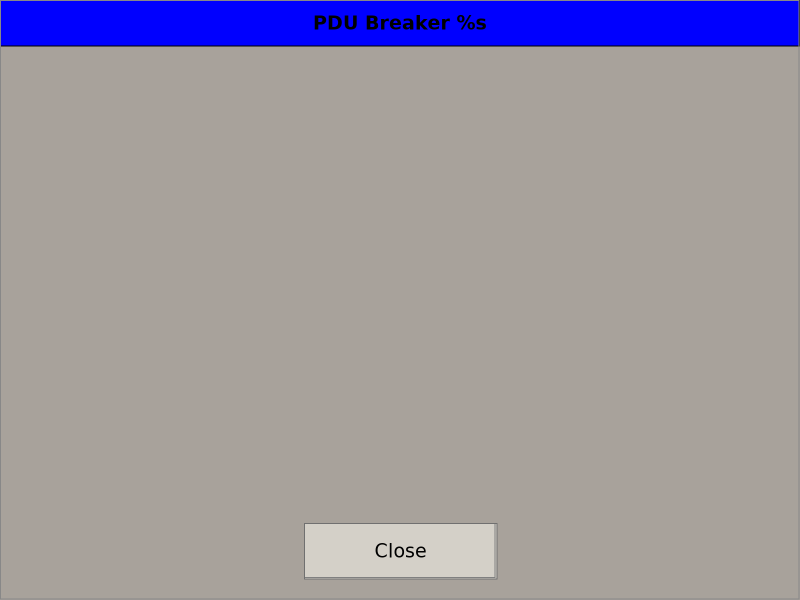
VISUALIZATION Dialog_PDU  // 800x600
VAR_IN_OUT
	sHeader : WSTRING;
	bCommonAlarm : BOOL;
	bIsolator1Alm :BOOL;
	bIsolator2Alm :BOOL;
END_VAR
    Rectangle (0,0 800x46), "PDU Breaker %s", text variable: sHeader
    Button (304,523 193x56), "Close"
        OnMouseClick: CloseDialog Dialog=Dialog_CRAH, Result=OK, NumpadKeypadSet=True
END_VISUALIZATION

(* stored: Version 1.1.0.1, ProductVersion 3.1.4024.12
   Visu Dialog_PDU: Id {0e983fc0-f887-4d24-b71b-0bad6634c7ef} *)
